FUNCTION_BLOCK FB_PowerAxis1
VAR
  stm	: UINT := 10;
  bFW, bBW,bPower,bReset,bResetDone,bError,bBusy,bPowerStatus : BOOL := FALSE;
  errId : UDINT;
  
  fbPower : MC_Power;
  fbReset : MC_Reset;
END_VAR

fbPower(
	Axis:= G.stAX.L1LeftFront, 
	Enable:= bPower, 
	Enable_Positive:= bPower, 
	Enable_Negative:= bPower, 
	Override:= 100.0, 
  Status=>bPowerStatus,
	Busy=>bBusy , 
	Error=>bError, 
	ErrorID=> errId);

fbReset(
	Axis:= G.stAX.L1LeftFront, 
	Execute:= bReset, 
	Done=> bResetDone,
	Busy=> bBusy, 
	Error=>bError, 
	ErrorID=>errId);
  
CASE stm OF 
  10:
		bPower := TRUE;
		stm := 20;
	20:
		IF G.stAX.L1LeftFront.Status.Error THEN //really at the level of NC
			stm := 30;
		ELSE
			stm := 50;
		END_IF
	30:
		bReset := TRUE;
		stm := 40;	
	40:
		IF bResetDone THEN
			bReset := FALSE;
			stm := 50;
		END_IF
	50:
    bPowerStatus := fbPower.Status;
		IF bPowerStatus THEN
			stm := 0;
		END_IF
   
  0:stm := 0;
END_CASE

END_FUNCTION_BLOCK

(* stored: Version 1.1.0.1, ProductVersion 3.1.4024.12
   POU FB_PowerAxis1: Id {0630e2cf-2446-4a55-9ef4-978bf9a13065}, SpecialFunc None *)
